{attribute 'qualified_only'}
VAR_GLOBAL CONSTANT
	{attribute 'OPC.UA.DA' := '0'}
	C_nNumAxes:	INT	:= 3;
END_VAR

(* stored: Version 1.1.0.1, ProductVersion 3.1.4022.16
   GVL GVL: Id {b3bf7d87-5e30-40ad-9919-75d8d50001fc} *)
